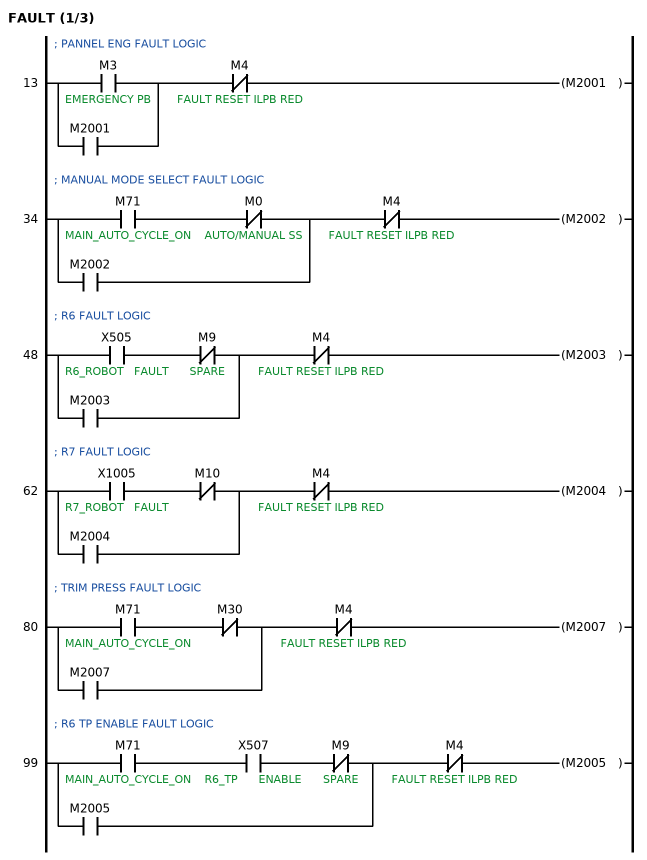
; PANNEL ENG FAULT LOGIC
13    LD      M3  ; EMERGENCY PB
      OR      M2001
      ANI     M4  ; FAULT RESET ILPB RED
      OUT     M2001
; MANUAL MODE SELECT FAULT LOGIC
34    LD      M71  ; MAIN_AUTO_CYCLE_ON
      ANI     M0  ; AUTO/MANUAL SS
      OR      M2002
      ANI     M4  ; FAULT RESET ILPB RED
      OUT     M2002
; R6 FAULT LOGIC
48    LD      X505  ; R6_ROBOT   FAULT
      ANI     M9  ; SPARE
      OR      M2003
      ANI     M4  ; FAULT RESET ILPB RED
      OUT     M2003
; R7 FAULT LOGIC
62    LD      X1005  ; R7_ROBOT   FAULT
      ANI     M10
      OR      M2004
      ANI     M4  ; FAULT RESET ILPB RED
      OUT     M2004
; TRIM PRESS FAULT LOGIC
80    LD      M71  ; MAIN_AUTO_CYCLE_ON
      ANI     M30
      OR      M2007
      ANI     M4  ; FAULT RESET ILPB RED
      OUT     M2007
; R6 TP ENABLE FAULT LOGIC
99    LD      M71  ; MAIN_AUTO_CYCLE_ON
      AND     X507  ; R6_TP      ENABLE
      ANI     M9  ; SPARE
      OR      M2005
      ANI     M4  ; FAULT RESET ILPB RED
      OUT     M2005
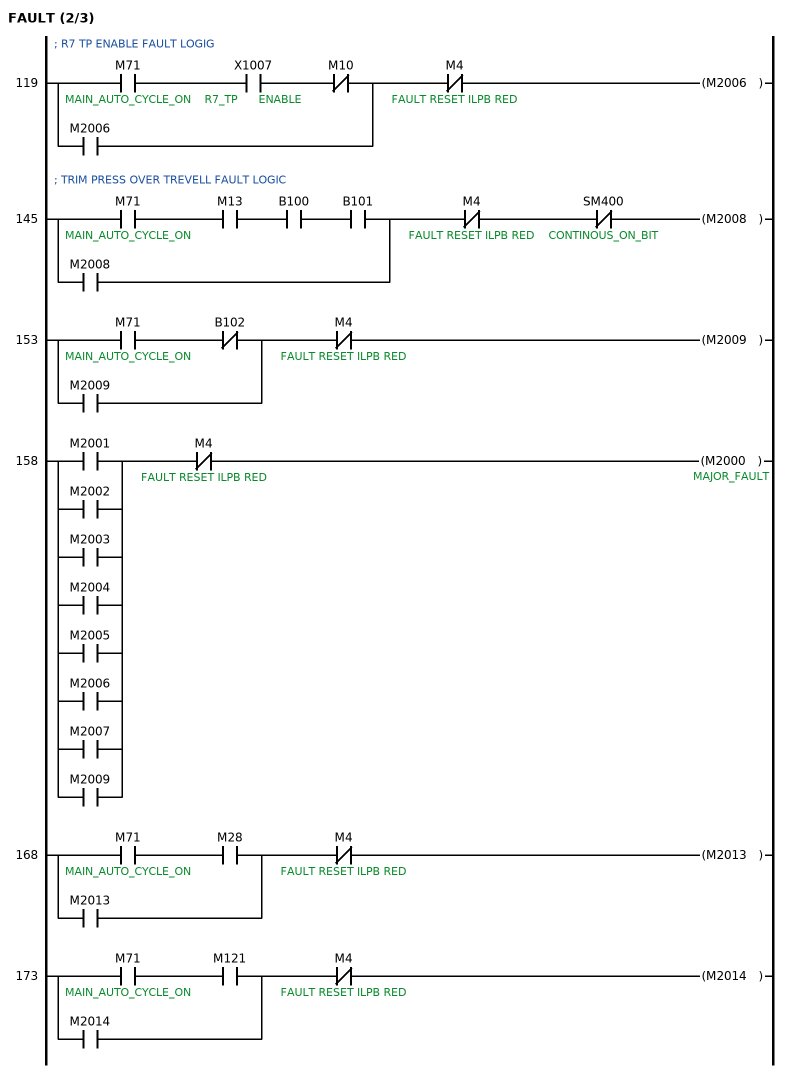
; R7 TP ENABLE FAULT LOGIG
119   LD      M71  ; MAIN_AUTO_CYCLE_ON
      AND     X1007  ; R7_TP      ENABLE
      ANI     M10
      OR      M2006
      ANI     M4  ; FAULT RESET ILPB RED
      OUT     M2006
; TRIM PRESS OVER TREVELL FAULT LOGIC
145   LD      M71  ; MAIN_AUTO_CYCLE_ON
      AND     M13
      AND     B100
      AND     B101
      OR      M2008
      ANI     M4  ; FAULT RESET ILPB RED
      ANI     SM400  ; CONTINOUS_ON_BIT
      OUT     M2008
153   LD      M71  ; MAIN_AUTO_CYCLE_ON
      ANI     B102
      OR      M2009
      ANI     M4  ; FAULT RESET ILPB RED
      OUT     M2009
158   LD      M2001
      OR      M2002
      OR      M2003
      OR      M2004
      OR      M2005
      OR      M2006
      OR      M2007
      OR      M2009
      ANI     M4  ; FAULT RESET ILPB RED
      OUT     M2000  ; MAJOR_FAULT
168   LD      M71  ; MAIN_AUTO_CYCLE_ON
      AND     M28
      OR      M2013
      ANI     M4  ; FAULT RESET ILPB RED
      OUT     M2013
173   LD      M71  ; MAIN_AUTO_CYCLE_ON
      AND     M121
      OR      M2014
      ANI     M4  ; FAULT RESET ILPB RED
      OUT     M2014
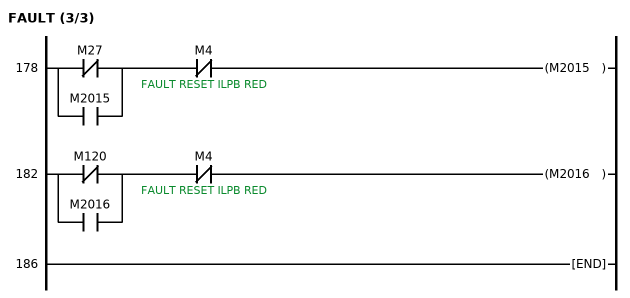
178   LDI     M27
      OR      M2015
      ANI     M4  ; FAULT RESET ILPB RED
      OUT     M2015
182   LDI     M120
      OR      M2016
      ANI     M4  ; FAULT RESET ILPB RED
      OUT     M2016
186   END
END_PROGRAM

PROGRAM ROBOT_3
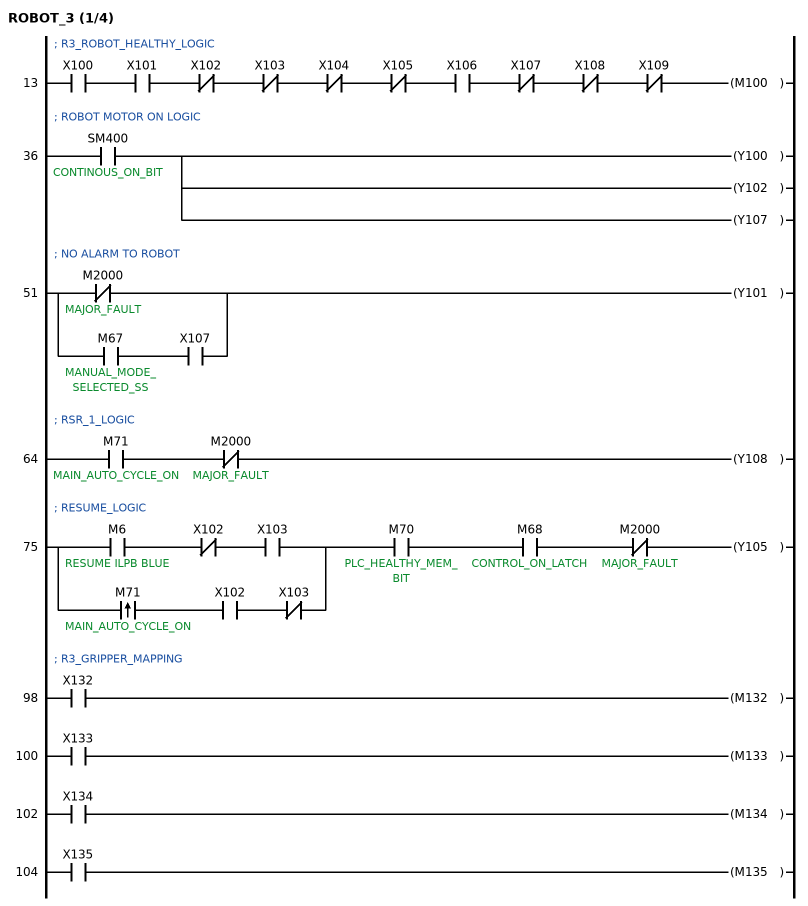
; R3_ROBOT_HEALTHY_LOGIC
13    LD      X100
      AND     X101
      ANI     X102
      ANI     X103
      ANI     X104
      ANI     X105
      AND     X106
      ANI     X107
      ANI     X108
      ANI     X109
      OUT     M100
; ROBOT MOTOR ON LOGIC
36    LD      SM400  ; CONTINOUS_ON_BIT
      OUT     Y100
      OUT     Y102
      OUT     Y107
; NO ALARM TO ROBOT
51    LDI     M2000  ; MAJOR_FAULT
      LD      M67  ; MANUAL_MODE_SELECTED_SS
      AND     X107
      ORB
      OUT     Y101
; RSR_1_LOGIC
64    LD      M71  ; MAIN_AUTO_CYCLE_ON
      ANI     M2000  ; MAJOR_FAULT
      OUT     Y108
; RESUME_LOGIC
75    LD      M6  ; RESUME ILPB BLUE
      ANI     X102
      AND     X103
      LDP     M71  ; MAIN_AUTO_CYCLE_ON
      AND     X102
      ANI     X103
      ORB
      AND     M70  ; PLC_HEALTHY_MEM_BIT
      AND     M68  ; CONTROL_ON_LATCH
      ANI     M2000  ; MAJOR_FAULT
      OUT     Y105
; R3_GRIPPER_MAPPING
98    LD      X132
      OUT     M132
100   LD      X133
      OUT     M133
102   LD      X134
      OUT     M134
104   LD      X135
      OUT     M135
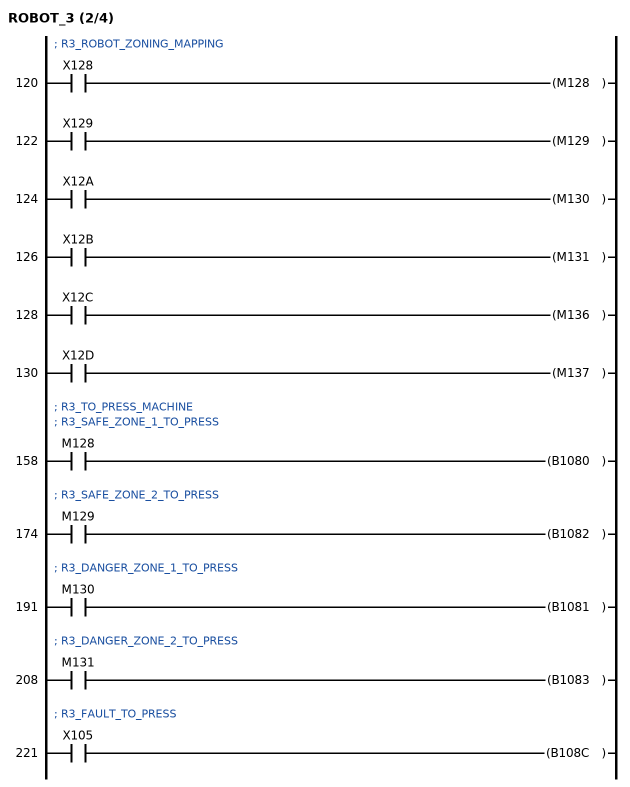
; R3_ROBOT_ZONING_MAPPING
120   LD      X128
      OUT     M128
122   LD      X129
      OUT     M129
124   LD      X12A
      OUT     M130
126   LD      X12B
      OUT     M131
128   LD      X12C
      OUT     M136
130   LD      X12D
      OUT     M137
; R3_TO_PRESS_MACHINE
; R3_SAFE_ZONE_1_TO_PRESS
158   LD      M128
      OUT     B1080
; R3_SAFE_ZONE_2_TO_PRESS
174   LD      M129
      OUT     B1082
; R3_DANGER_ZONE_1_TO_PRESS
191   LD      M130
      OUT     B1081
; R3_DANGER_ZONE_2_TO_PRESS
208   LD      M131
      OUT     B1083
; R3_FAULT_TO_PRESS
221   LD      X105
      OUT     B108C
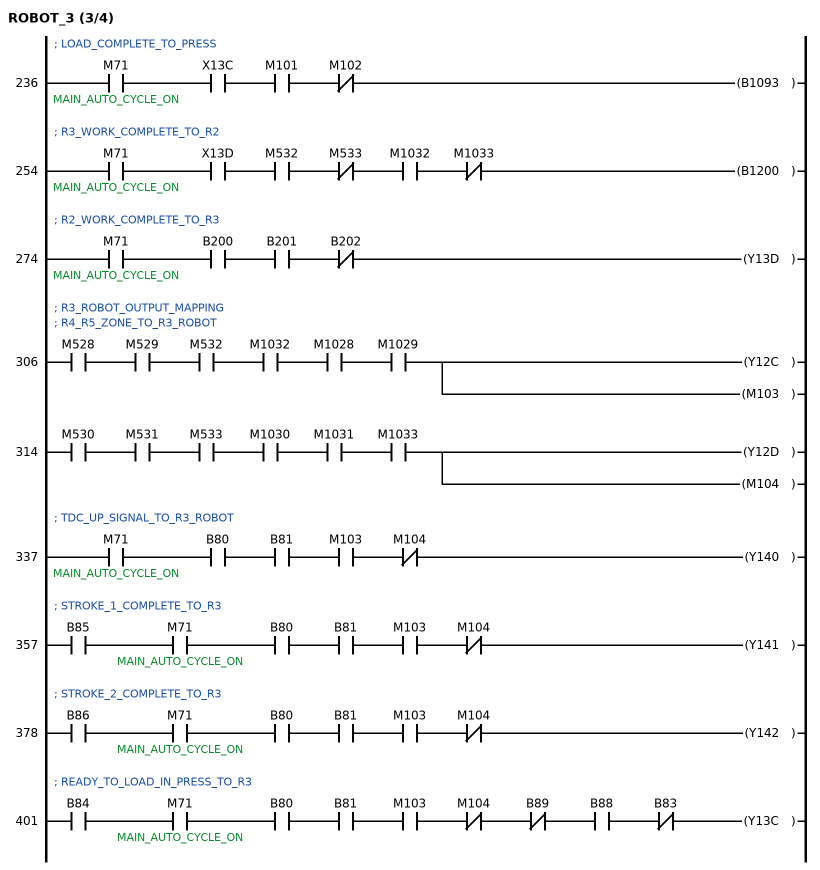
; LOAD_COMPLETE_TO_PRESS
236   LD      M71  ; MAIN_AUTO_CYCLE_ON
      AND     X13C
      AND     M101
      ANI     M102
      OUT     B1093
; R3_WORK_COMPLETE_TO_R2
254   LD      M71  ; MAIN_AUTO_CYCLE_ON
      AND     X13D
      AND     M532
      ANI     M533
      AND     M1032
      ANI     M1033
      OUT     B1200
; R2_WORK_COMPLETE_TO_R3
274   LD      M71  ; MAIN_AUTO_CYCLE_ON
      AND     B200
      AND     B201
      ANI     B202
      OUT     Y13D
; R3_ROBOT_OUTPUT_MAPPING
; R4_R5_ZONE_TO_R3_ROBOT
306   LD      M528
      AND     M529
      AND     M532
      AND     M1032
      AND     M1028
      AND     M1029
      OUT     Y12C
      OUT     M103
314   LD      M530
      AND     M531
      AND     M533
      AND     M1030
      AND     M1031
      AND     M1033
      OUT     Y12D
      OUT     M104
; TDC_UP_SIGNAL_TO_R3_ROBOT
337   LD      M71  ; MAIN_AUTO_CYCLE_ON
      AND     B80
      AND     B81
      AND     M103
      ANI     M104
      OUT     Y140
; STROKE_1_COMPLETE_TO_R3
357   LD      B85
      AND     M71  ; MAIN_AUTO_CYCLE_ON
      AND     B80
      AND     B81
      AND     M103
      ANI     M104
      OUT     Y141
; STROKE_2_COMPLETE_TO_R3
378   LD      B86
      AND     M71  ; MAIN_AUTO_CYCLE_ON
      AND     B80
      AND     B81
      AND     M103
      ANI     M104
      OUT     Y142
; READY_TO_LOAD_IN_PRESS_TO_R3
401   LD      B84
      AND     M71  ; MAIN_AUTO_CYCLE_ON
      AND     B80
      AND     B81
      AND     M103
      ANI     M104
      ANI     B89
      AND     B88
      ANI     B83
      OUT     Y13C
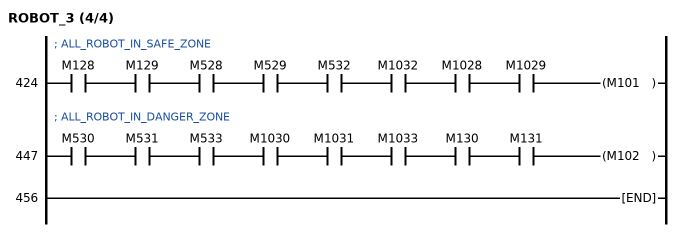
; ALL_ROBOT_IN_SAFE_ZONE
424   LD      M128
      AND     M129
      AND     M528
      AND     M529
      AND     M532
      AND     M1032
      AND     M1028
      AND     M1029
      OUT     M101
; ALL_ROBOT_IN_DANGER_ZONE
447   LD      M530
      AND     M531
      AND     M533
      AND     M1030
      AND     M1031
      AND     M1033
      AND     M130
      AND     M131
      OUT     M102
456   END
END_PROGRAM

PROGRAM ROBOT_4
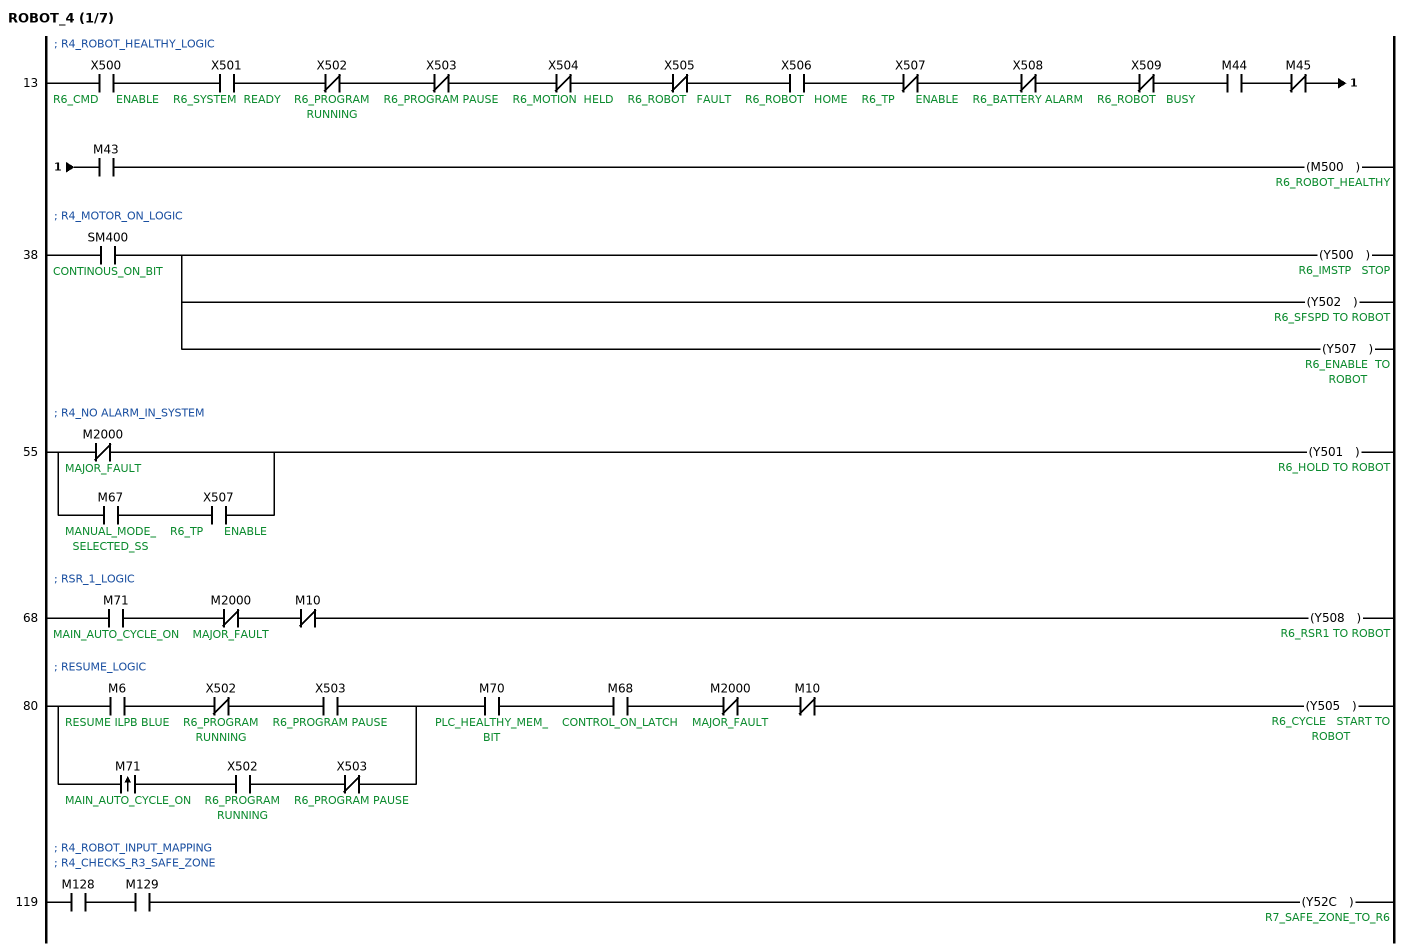
; R4_ROBOT_HEALTHY_LOGIC
13    LD      X500  ; R6_CMD     ENABLE
      AND     X501  ; R6_SYSTEM  READY
      ANI     X502  ; R6_PROGRAM RUNNING
      ANI     X503  ; R6_PROGRAM PAUSE
      ANI     X504  ; R6_MOTION  HELD
      ANI     X505  ; R6_ROBOT   FAULT
      AND     X506  ; R6_ROBOT   HOME
      ANI     X507  ; R6_TP      ENABLE
      ANI     X508  ; R6_BATTERY ALARM
      ANI     X509  ; R6_ROBOT   BUSY
      AND     M44
      ANI     M45
      AND     M43
      OUT     M500  ; R6_ROBOT_HEALTHY
; R4_MOTOR_ON_LOGIC
38    LD      SM400  ; CONTINOUS_ON_BIT
      OUT     Y500  ; R6_IMSTP   STOP
      OUT     Y502  ; R6_SFSPD TO ROBOT
      OUT     Y507  ; R6_ENABLE  TO ROBOT
; R4_NO ALARM_IN_SYSTEM
55    LDI     M2000  ; MAJOR_FAULT
      LD      M67  ; MANUAL_MODE_SELECTED_SS
      AND     X507  ; R6_TP      ENABLE
      ORB
      OUT     Y501  ; R6_HOLD TO ROBOT
; RSR_1_LOGIC
68    LD      M71  ; MAIN_AUTO_CYCLE_ON
      ANI     M2000  ; MAJOR_FAULT
      ANI     M10
      OUT     Y508  ; R6_RSR1 TO ROBOT
; RESUME_LOGIC
80    LD      M6  ; RESUME ILPB BLUE
      ANI     X502  ; R6_PROGRAM RUNNING
      AND     X503  ; R6_PROGRAM PAUSE
      LDP     M71  ; MAIN_AUTO_CYCLE_ON
      AND     X502  ; R6_PROGRAM RUNNING
      ANI     X503  ; R6_PROGRAM PAUSE
      ORB
      AND     M70  ; PLC_HEALTHY_MEM_BIT
      AND     M68  ; CONTROL_ON_LATCH
      ANI     M2000  ; MAJOR_FAULT
      ANI     M10
      OUT     Y505  ; R6_CYCLE   START TO ROBOT
; R4_ROBOT_INPUT_MAPPING
; R4_CHECKS_R3_SAFE_ZONE
119   LD      M128
      AND     M129
      OUT     Y52C  ; R7_SAFE_ZONE_TO_R6
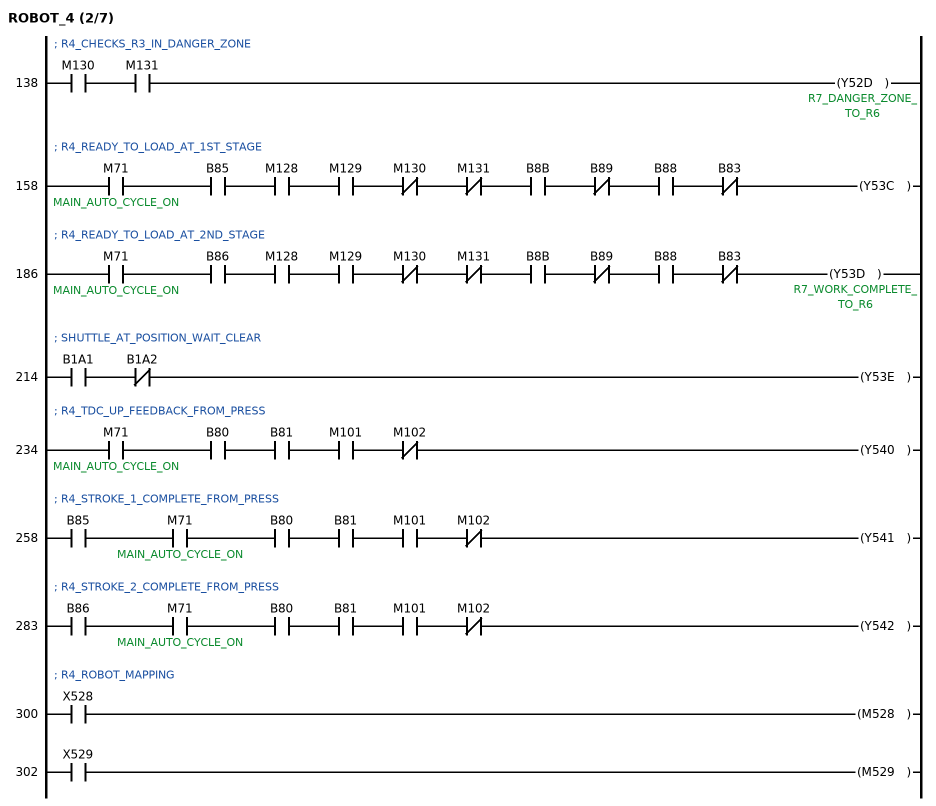
; R4_CHECKS_R3_IN_DANGER_ZONE
138   LD      M130
      AND     M131
      OUT     Y52D  ; R7_DANGER_ZONE_TO_R6
; R4_READY_TO_LOAD_AT_1ST_STAGE
158   LD      M71  ; MAIN_AUTO_CYCLE_ON
      AND     B85
      AND     M128
      AND     M129
      ANI     M130
      ANI     M131
      AND     B8B
      ANI     B89
      AND     B88
      ANI     B83
      OUT     Y53C
; R4_READY_TO_LOAD_AT_2ND_STAGE
186   LD      M71  ; MAIN_AUTO_CYCLE_ON
      AND     B86
      AND     M128
      AND     M129
      ANI     M130
      ANI     M131
      AND     B8B
      ANI     B89
      AND     B88
      ANI     B83
      OUT     Y53D  ; R7_WORK_COMPLETE_TO_R6
; SHUTTLE_AT_POSITION_WAIT_CLEAR
214   LD      B1A1
      ANI     B1A2
      OUT     Y53E
; R4_TDC_UP_FEEDBACK_FROM_PRESS
234   LD      M71  ; MAIN_AUTO_CYCLE_ON
      AND     B80
      AND     B81
      AND     M101
      ANI     M102
      OUT     Y540
; R4_STROKE_1_COMPLETE_FROM_PRESS
258   LD      B85
      AND     M71  ; MAIN_AUTO_CYCLE_ON
      AND     B80
      AND     B81
      AND     M101
      ANI     M102
      OUT     Y541
; R4_STROKE_2_COMPLETE_FROM_PRESS
283   LD      B86
      AND     M71  ; MAIN_AUTO_CYCLE_ON
      AND     B80
      AND     B81
      AND     M101
      ANI     M102
      OUT     Y542
; R4_ROBOT_MAPPING
300   LD      X528
      OUT     M528
302   LD      X529
      OUT     M529
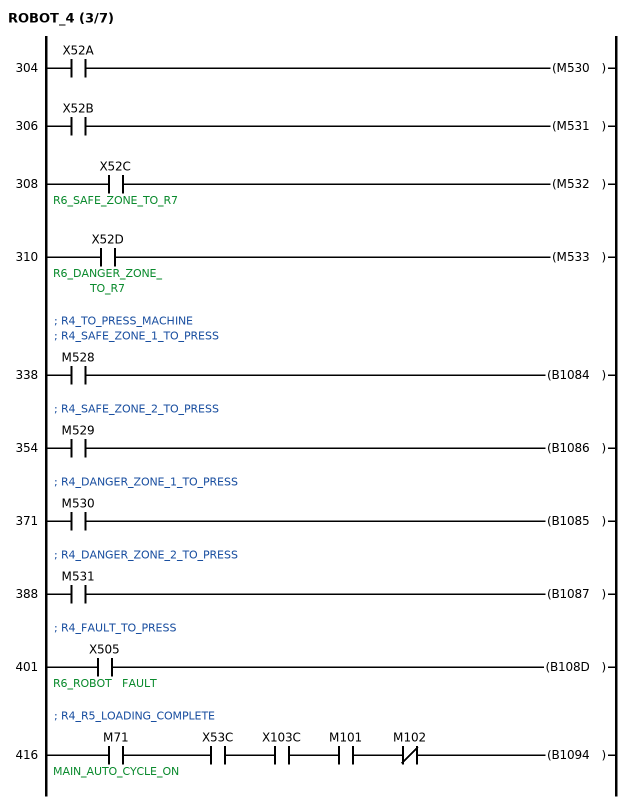
304   LD      X52A
      OUT     M530
306   LD      X52B
      OUT     M531
308   LD      X52C  ; R6_SAFE_ZONE_TO_R7
      OUT     M532
310   LD      X52D  ; R6_DANGER_ZONE_TO_R7
      OUT     M533
; R4_TO_PRESS_MACHINE
; R4_SAFE_ZONE_1_TO_PRESS
338   LD      M528
      OUT     B1084
; R4_SAFE_ZONE_2_TO_PRESS
354   LD      M529
      OUT     B1086
; R4_DANGER_ZONE_1_TO_PRESS
371   LD      M530
      OUT     B1085
; R4_DANGER_ZONE_2_TO_PRESS
388   LD      M531
      OUT     B1087
; R4_FAULT_TO_PRESS
401   LD      X505  ; R6_ROBOT   FAULT
      OUT     B108D
; R4_R5_LOADING_COMPLETE
416   LD      M71  ; MAIN_AUTO_CYCLE_ON
      AND     X53C
      AND     X103C
      AND     M101
      ANI     M102
      OUT     B1094
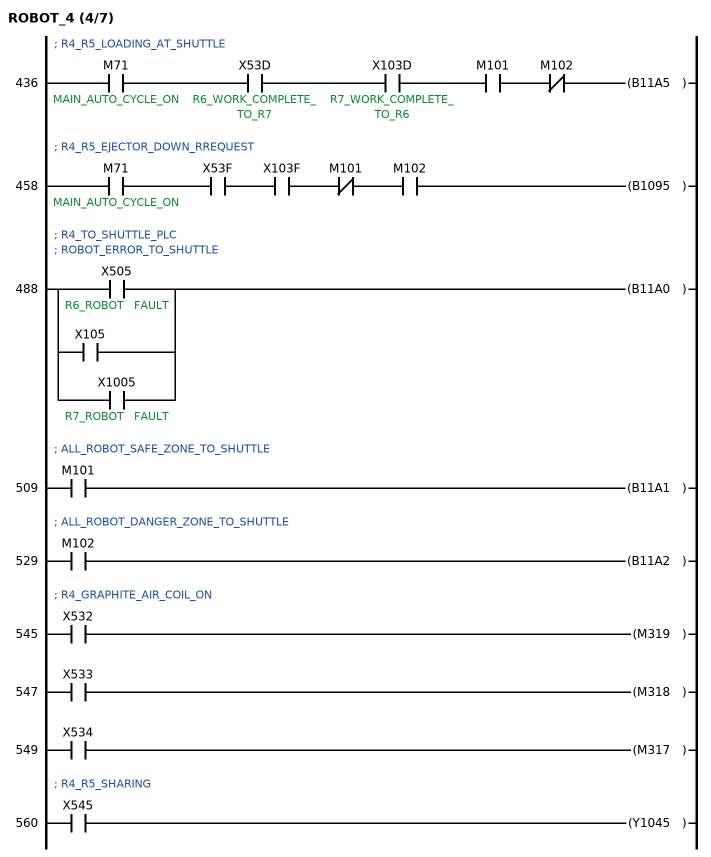
; R4_R5_LOADING_AT_SHUTTLE
436   LD      M71  ; MAIN_AUTO_CYCLE_ON
      AND     X53D  ; R6_WORK_COMPLETE_TO_R7
      AND     X103D  ; R7_WORK_COMPLETE_TO_R6
      AND     M101
      ANI     M102
      OUT     B11A5
; R4_R5_EJECTOR_DOWN_RREQUEST
458   LD      M71  ; MAIN_AUTO_CYCLE_ON
      AND     X53F
      AND     X103F
      ANI     M101
      AND     M102
      OUT     B1095
; R4_TO_SHUTTLE_PLC
; ROBOT_ERROR_TO_SHUTTLE
488   LD      X505  ; R6_ROBOT   FAULT
      OR      X105
      OR      X1005  ; R7_ROBOT   FAULT
      OUT     B11A0
; ALL_ROBOT_SAFE_ZONE_TO_SHUTTLE
509   LD      M101
      OUT     B11A1
; ALL_ROBOT_DANGER_ZONE_TO_SHUTTLE
529   LD      M102
      OUT     B11A2
; R4_GRAPHITE_AIR_COIL_ON
545   LD      X532
      OUT     M319
547   LD      X533
      OUT     M318
549   LD      X534
      OUT     M317
; R4_R5_SHARING
560   LD      X545
      OUT     Y1045
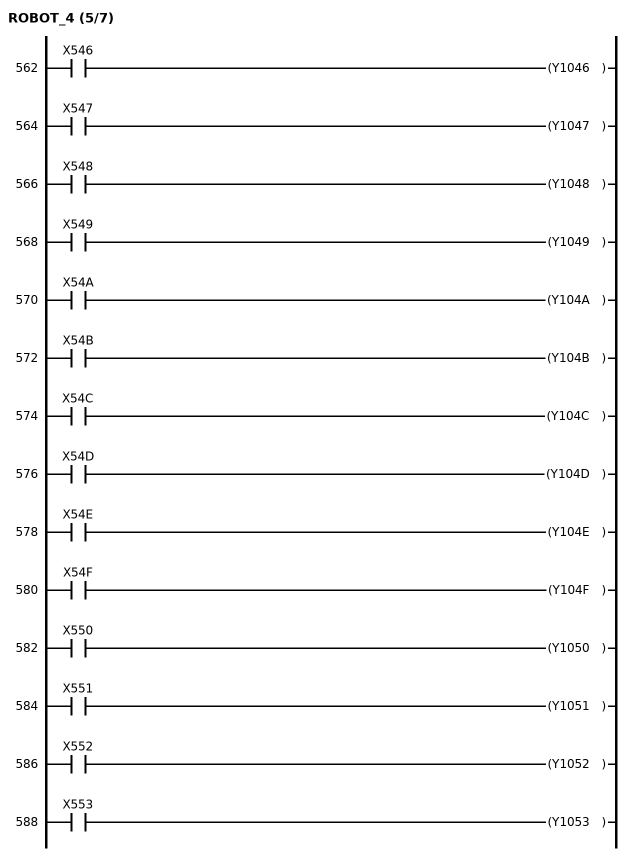
562   LD      X546
      OUT     Y1046
564   LD      X547
      OUT     Y1047
566   LD      X548
      OUT     Y1048
568   LD      X549
      OUT     Y1049
570   LD      X54A
      OUT     Y104A
572   LD      X54B
      OUT     Y104B
574   LD      X54C
      OUT     Y104C
576   LD      X54D
      OUT     Y104D
578   LD      X54E
      OUT     Y104E
580   LD      X54F
      OUT     Y104F
582   LD      X550
      OUT     Y1050
584   LD      X551
      OUT     Y1051
586   LD      X552
      OUT     Y1052
588   LD      X553
      OUT     Y1053
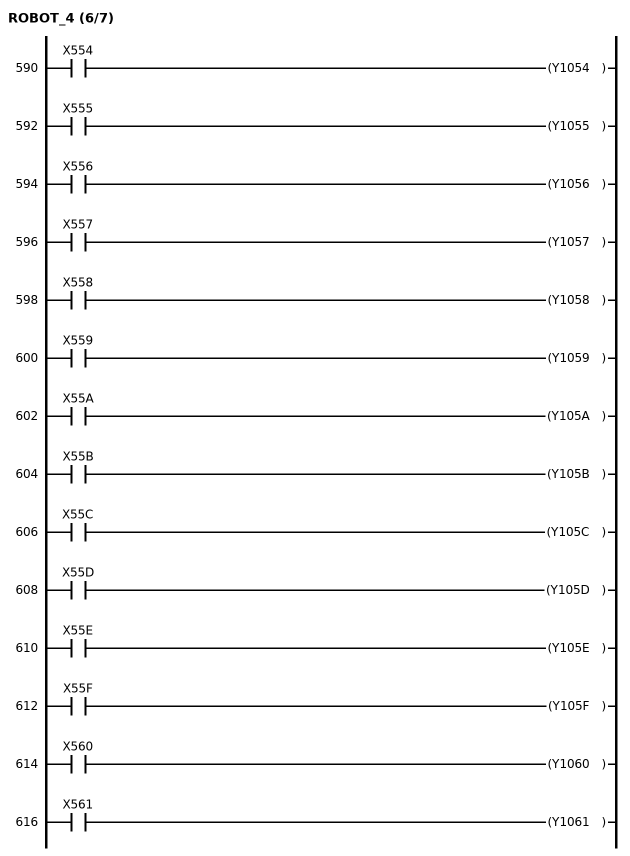
590   LD      X554
      OUT     Y1054
592   LD      X555
      OUT     Y1055
594   LD      X556
      OUT     Y1056
596   LD      X557
      OUT     Y1057
598   LD      X558
      OUT     Y1058
600   LD      X559
      OUT     Y1059
602   LD      X55A
      OUT     Y105A
604   LD      X55B
      OUT     Y105B
606   LD      X55C
      OUT     Y105C
608   LD      X55D
      OUT     Y105D
610   LD      X55E
      OUT     Y105E
612   LD      X55F
      OUT     Y105F
614   LD      X560
      OUT     Y1060
616   LD      X561
      OUT     Y1061
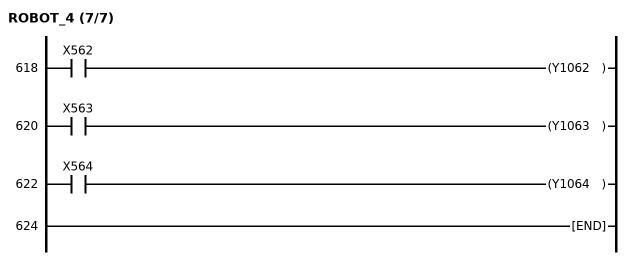
618   LD      X562
      OUT     Y1062
620   LD      X563
      OUT     Y1063
622   LD      X564
      OUT     Y1064
624   END
END_PROGRAM

PROGRAM ROBOT_5
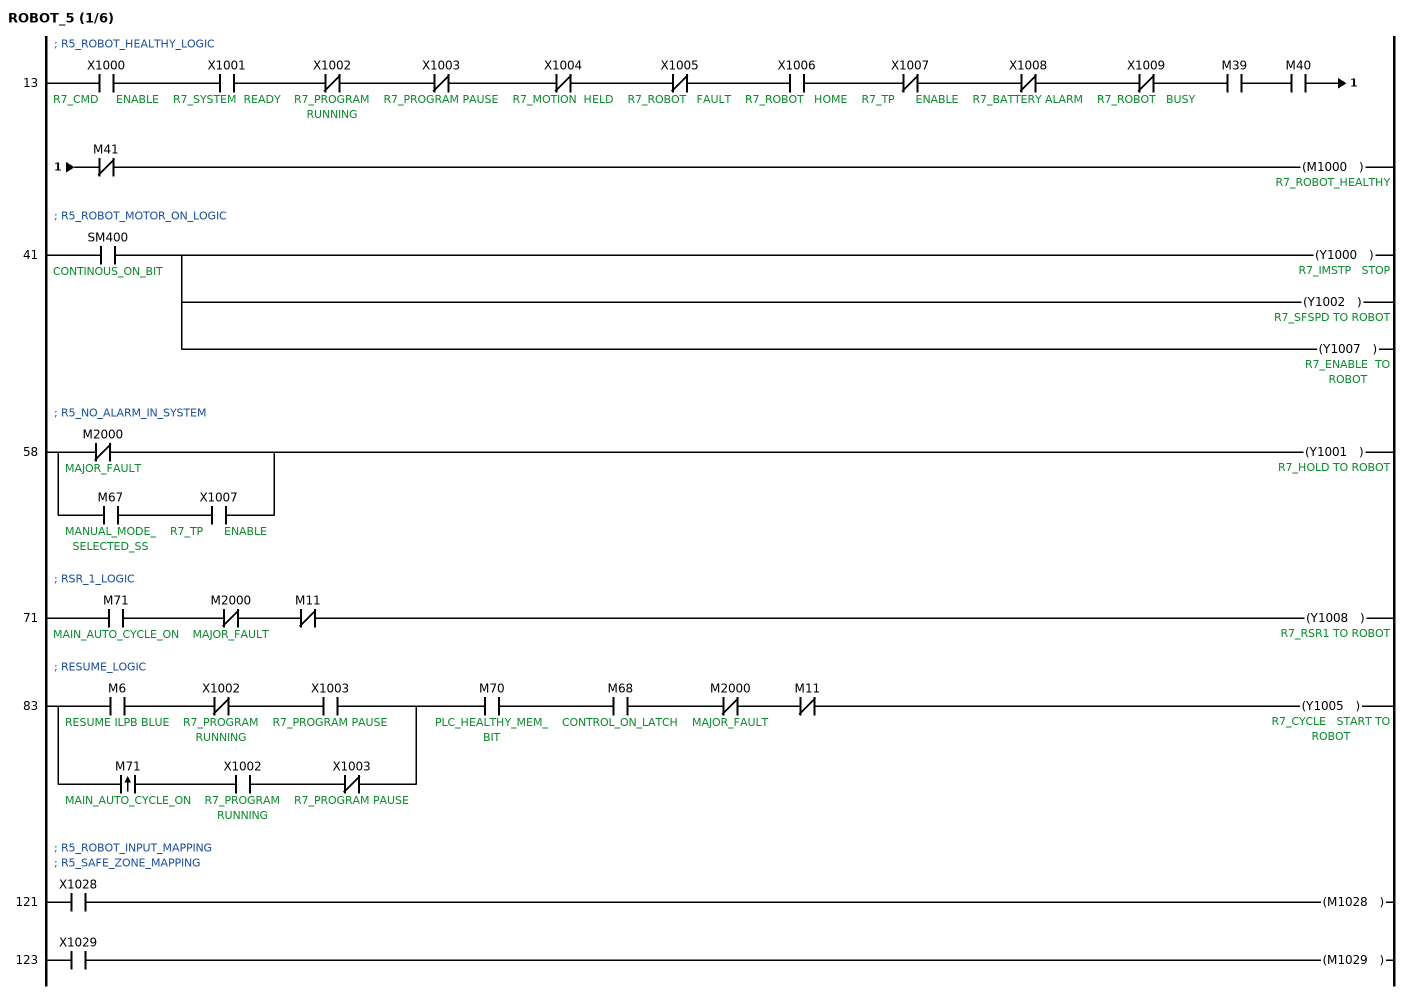
; R5_ROBOT_HEALTHY_LOGIC
13    LD      X1000  ; R7_CMD     ENABLE
      AND     X1001  ; R7_SYSTEM  READY
      ANI     X1002  ; R7_PROGRAM RUNNING
      ANI     X1003  ; R7_PROGRAM PAUSE
      ANI     X1004  ; R7_MOTION  HELD
      ANI     X1005  ; R7_ROBOT   FAULT
      AND     X1006  ; R7_ROBOT   HOME
      ANI     X1007  ; R7_TP      ENABLE
      ANI     X1008  ; R7_BATTERY ALARM
      ANI     X1009  ; R7_ROBOT   BUSY
      AND     M39
      AND     M40
      ANI     M41
      OUT     M1000  ; R7_ROBOT_HEALTHY
; R5_ROBOT_MOTOR_ON_LOGIC
41    LD      SM400  ; CONTINOUS_ON_BIT
      OUT     Y1000  ; R7_IMSTP   STOP
      OUT     Y1002  ; R7_SFSPD TO ROBOT
      OUT     Y1007  ; R7_ENABLE  TO ROBOT
; R5_NO_ALARM_IN_SYSTEM
58    LDI     M2000  ; MAJOR_FAULT
      LD      M67  ; MANUAL_MODE_SELECTED_SS
      AND     X1007  ; R7_TP      ENABLE
      ORB
      OUT     Y1001  ; R7_HOLD TO ROBOT
; RSR_1_LOGIC
71    LD      M71  ; MAIN_AUTO_CYCLE_ON
      ANI     M2000  ; MAJOR_FAULT
      ANI     M11
      OUT     Y1008  ; R7_RSR1 TO ROBOT
; RESUME_LOGIC
83    LD      M6  ; RESUME ILPB BLUE
      ANI     X1002  ; R7_PROGRAM RUNNING
      AND     X1003  ; R7_PROGRAM PAUSE
      LDP     M71  ; MAIN_AUTO_CYCLE_ON
      AND     X1002  ; R7_PROGRAM RUNNING
      ANI     X1003  ; R7_PROGRAM PAUSE
      ORB
      AND     M70  ; PLC_HEALTHY_MEM_BIT
      AND     M68  ; CONTROL_ON_LATCH
      ANI     M2000  ; MAJOR_FAULT
      ANI     M11
      OUT     Y1005  ; R7_CYCLE   START TO ROBOT
; R5_ROBOT_INPUT_MAPPING
; R5_SAFE_ZONE_MAPPING
121   LD      X1028
      OUT     M1028
123   LD      X1029
      OUT     M1029
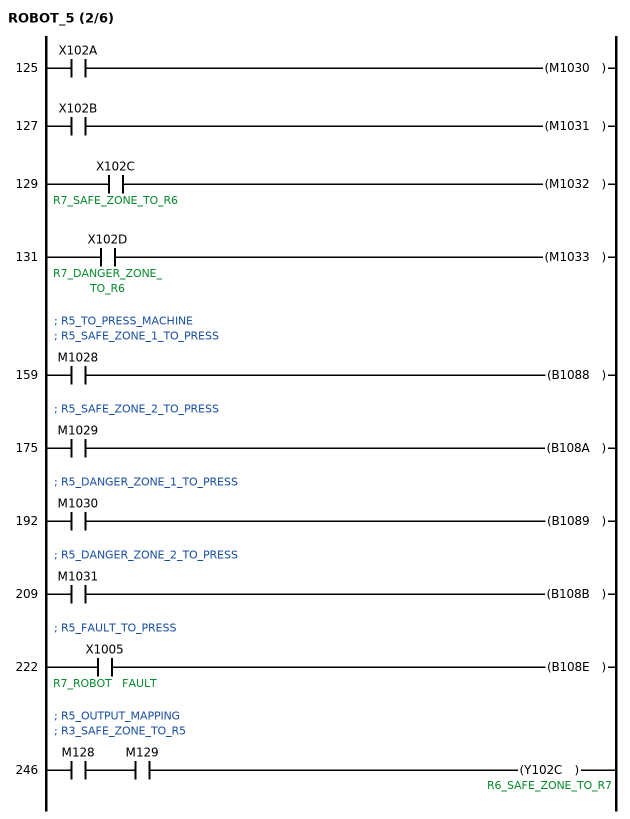
125   LD      X102A
      OUT     M1030
127   LD      X102B
      OUT     M1031
129   LD      X102C  ; R7_SAFE_ZONE_TO_R6
      OUT     M1032
131   LD      X102D  ; R7_DANGER_ZONE_TO_R6
      OUT     M1033
; R5_TO_PRESS_MACHINE
; R5_SAFE_ZONE_1_TO_PRESS
159   LD      M1028
      OUT     B1088
; R5_SAFE_ZONE_2_TO_PRESS
175   LD      M1029
      OUT     B108A
; R5_DANGER_ZONE_1_TO_PRESS
192   LD      M1030
      OUT     B1089
; R5_DANGER_ZONE_2_TO_PRESS
209   LD      M1031
      OUT     B108B
; R5_FAULT_TO_PRESS
222   LD      X1005  ; R7_ROBOT   FAULT
      OUT     B108E
; R5_OUTPUT_MAPPING
; R3_SAFE_ZONE_TO_R5
246   LD      M128
      AND     M129
      OUT     Y102C  ; R6_SAFE_ZONE_TO_R7
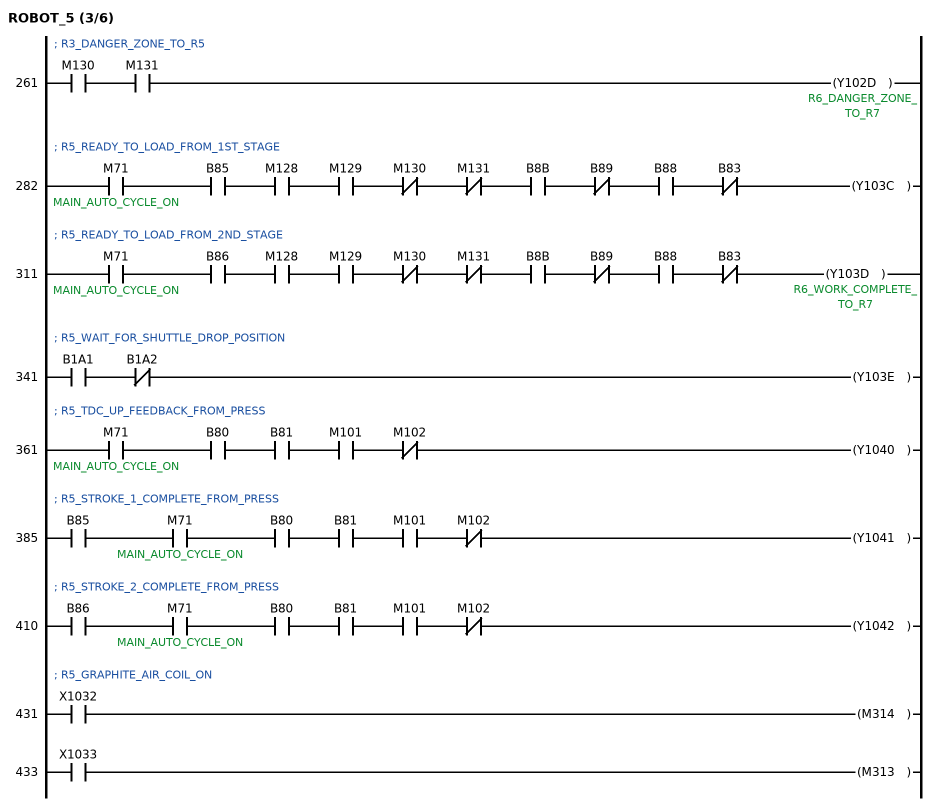
; R3_DANGER_ZONE_TO_R5
261   LD      M130
      AND     M131
      OUT     Y102D  ; R6_DANGER_ZONE_TO_R7
; R5_READY_TO_LOAD_FROM_1ST_STAGE
282   LD      M71  ; MAIN_AUTO_CYCLE_ON
      AND     B85
      AND     M128
      AND     M129
      ANI     M130
      ANI     M131
      AND     B8B
      ANI     B89
      AND     B88
      ANI     B83
      OUT     Y103C
; R5_READY_TO_LOAD_FROM_2ND_STAGE
311   LD      M71  ; MAIN_AUTO_CYCLE_ON
      AND     B86
      AND     M128
      AND     M129
      ANI     M130
      ANI     M131
      AND     B8B
      ANI     B89
      AND     B88
      ANI     B83
      OUT     Y103D  ; R6_WORK_COMPLETE_TO_R7
; R5_WAIT_FOR_SHUTTLE_DROP_POSITION
341   LD      B1A1
      ANI     B1A2
      OUT     Y103E
; R5_TDC_UP_FEEDBACK_FROM_PRESS
361   LD      M71  ; MAIN_AUTO_CYCLE_ON
      AND     B80
      AND     B81
      AND     M101
      ANI     M102
      OUT     Y1040
; R5_STROKE_1_COMPLETE_FROM_PRESS
385   LD      B85
      AND     M71  ; MAIN_AUTO_CYCLE_ON
      AND     B80
      AND     B81
      AND     M101
      ANI     M102
      OUT     Y1041
; R5_STROKE_2_COMPLETE_FROM_PRESS
410   LD      B86
      AND     M71  ; MAIN_AUTO_CYCLE_ON
      AND     B80
      AND     B81
      AND     M101
      ANI     M102
      OUT     Y1042
; R5_GRAPHITE_AIR_COIL_ON
431   LD      X1032
      OUT     M314
433   LD      X1033
      OUT     M313
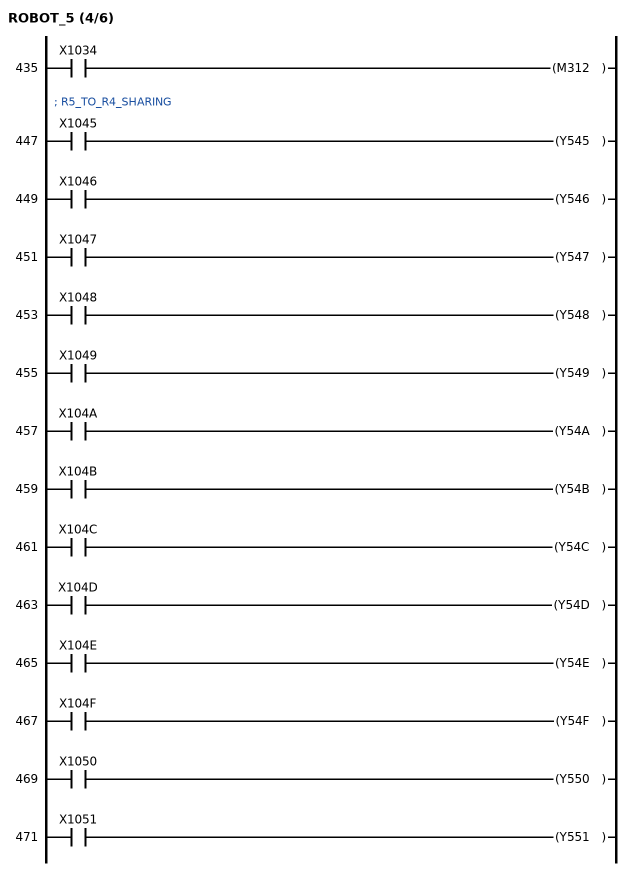
435   LD      X1034
      OUT     M312
; R5_TO_R4_SHARING
447   LD      X1045
      OUT     Y545
449   LD      X1046
      OUT     Y546
451   LD      X1047
      OUT     Y547
453   LD      X1048
      OUT     Y548
455   LD      X1049
      OUT     Y549
457   LD      X104A
      OUT     Y54A
459   LD      X104B
      OUT     Y54B
461   LD      X104C
      OUT     Y54C
463   LD      X104D
      OUT     Y54D
465   LD      X104E
      OUT     Y54E
467   LD      X104F
      OUT     Y54F
469   LD      X1050
      OUT     Y550
471   LD      X1051
      OUT     Y551
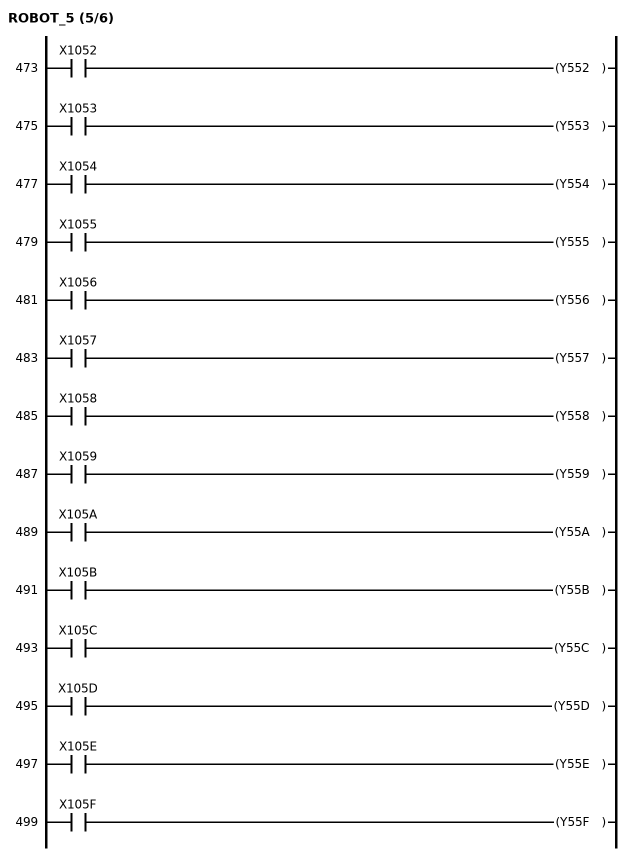
473   LD      X1052
      OUT     Y552
475   LD      X1053
      OUT     Y553
477   LD      X1054
      OUT     Y554
479   LD      X1055
      OUT     Y555
481   LD      X1056
      OUT     Y556
483   LD      X1057
      OUT     Y557
485   LD      X1058
      OUT     Y558
487   LD      X1059
      OUT     Y559
489   LD      X105A
      OUT     Y55A
491   LD      X105B
      OUT     Y55B
493   LD      X105C
      OUT     Y55C
495   LD      X105D
      OUT     Y55D
497   LD      X105E
      OUT     Y55E
499   LD      X105F
      OUT     Y55F
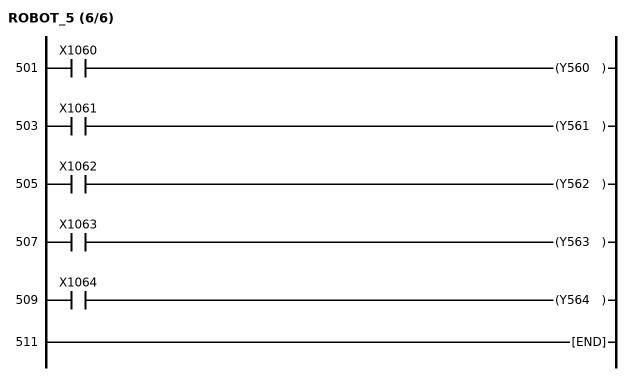
501   LD      X1060
      OUT     Y560
503   LD      X1061
      OUT     Y561
505   LD      X1062
      OUT     Y562
507   LD      X1063
      OUT     Y563
509   LD      X1064
      OUT     Y564
511   END
END_PROGRAM

// device comments not shown above
X50A  ; R6_ACK_1
X50B  ; R6_ACK_2
X50C  ; R6_ACK_3
X50D  ; R6_ACK_4
X50E  ; R6_ACK_5
X50F  ; R6_ACK_6
X510  ; R6_ACK_7
X511  ; R6_ACK_8
X512  ; R6_SNACK
X100A  ; R7_ACK_1
X100B  ; R7_ACK_2
X100C  ; R7_ACK_3
X100D  ; R7_ACK_4
X100E  ; R7_ACK_5
X100F  ; R7_ACK_6
X1010  ; R7_ACK_7
X1011  ; R7_ACK_8
X1012  ; R7_SNACK
Y43  ; CYCLE RESUME ILPB
Y503  ; R6_CYCLE   STOP TO ROBOT
Y506  ; R6_ROBOT   HOME TO ROBOT
Y509  ; R6_RSR2 TO ROBOT
Y50A  ; R6_RSR3 TO ROBOT
Y50B  ; R6_RSR4 TO ROBOT
Y50C  ; R6_RSR5 TO ROBOT
Y50D  ; R6_RSR6 TO ROBOT
Y50E  ; R6_RSR7 TO ROBOT
Y50F  ; R6_RSR8 TO ROBOT
Y510  ; R6_PNS     STROBE
Y511  ; R6_PRODUCTION START
Y1003  ; R7_CYCLE   STOP TO ROBOT
Y1006  ; R7_ROBOT   HOME TO ROBOT
Y1009  ; R7_RSR2 TO ROBOT
Y100A  ; R7_RSR3 TO ROBOT
Y100B  ; R7_RSR4 TO ROBOT
Y100C  ; R7_RSR5 TO ROBOT
Y100D  ; R7_RSR6 TO ROBOT
Y100E  ; R7_RSR7 TO ROBOT
Y100F  ; R7_RSR8 TO ROBOT
Y1010  ; R7_PNS     STROBE
Y1011  ; R7_PRODUCTION START
B1000  ; TDC1  TO PLC 2
B1001  ; TDC2  TO PLC 2
B1002  ; TRIM PRESS NO ERROR TO PLC 2
B1003  ; TRIM PRESS READY TO PLC 2
B1004  ; READY TO LOAD/UNLOAD SIGNAL TO P
B1021  ; SHUTTLE AT UNLOAD POSN TO PLC 2
B1022  ; SHUTTLE IN MOTION TO PLC 2
B1023  ; ROBOT R4 & R5 NO ERROR TO PLC 2
B1024  ; HMD TO PLC 2
